// TIA Portal V18 export
// export: Created 2025-12-01T12:39:35.9659709Z, ExportSetting None, DisplayName Totally Integrated Automation Portal, DisplayVersion V18 Update 5, DisplayName TIA Portal Openness, DisplayVersion V18 Update 5, DisplayName TIA Portal Teamcenter Gateway, DisplayVersion V18, DisplayName TIA Portal Version Control Interface, DisplayVersion V18, DisplayName STEP 7 Professional, DisplayVersion V18 Update 5, DisplayName STEP 7 Safety, DisplayVersion V18, DisplayName WinCC Professional, DisplayVersion V18 Update 5
VAR_GLOBAL   // PLC tag table "Lifting"
END_VAR
VAR_GLOBAL CONSTANT   // user constants
   Job_Run_in : Int := 10;   // 进料任务分配中
   Job_Run_out : Int := 15;   // 出料任务分配中
   Job_Run : Int := 60;   // 有任务在提升机运行
   Job_Run_in_done : Int := 11;   // 进料任务完成
   Job_Run_out_done : Int := 16;   // 出料任务完成
   Liftinghavepart : Int := 66;   // 提升机有托盘
END_VAR
